# EPICS IOC start-up script: tests/UTEST_IOC01/startup.iocsh
require iocStats
